Staubli VAL3: Apilar.dtx

bool bTraslada = true
bool bFin
bool bPiezaPreparada
bool bTermina
frame fTrabajo = {x=-400, y=175, z=-274.326706, fatherId=world[0]}
jointRx jHome
public mdesc mNomSpeed = {leave=25, reach=25}
mdesc mVelAprox = {accel=25, vel=50, decel=25, blend=off}
num nPiezaActual = 1
num nTrasladadas = 7
num nPiezaAltura = 12
num nSeparacion = 100
num nTotalPiezas = 2
pointRx p0 = {ry=180, fatherId=fTrabajo[0]}
pointRx pCentro = {x=-400, y=175, z=-272, ry=180, shoulder=righty, elbow=enegative, wrist=wnegative, fatherId=world[0]}
pointRx pDestino = {x=-2.694223E-15, y=50, z=22, rx=-180, ry=7.016709E-15, rz=-180, fatherId=fTrabajo[0]}
pointRx pEntrada = {y=-50, z=103, rx=-180, rz=-180, fatherId=fTrabajo[0]}
pointRx pOrigen = {x=-1.347111E-15, y=-50, z=11, rx=-180, ry=7.016709E-15, rz=-180, fatherId=fTrabajo[0]}
pointRx pEspera = {x=-6.123234E-15, z=50, rx=-180, ry=7.016709E-15, rz=-180, fatherId=fTrabajo[0]}
pointRx pSalida = {x=-1.347111E-15, y=50, z=11, rx=-180, ry=7.016709E-15, rz=-180, fatherId=fTrabajo[0]}
tool tEyector = {z=22, fatherId=flange[0], ioLink=valve1, ioOpen=1, ioClose=1}
trsf trAprox = {z=-50}
num nEspera
num nOffset
bool bHaciaSalida
pointRx pInicio = {fatherId=world[0]}
